// TIA Portal V19 export
VAR_GLOBAL   // PLC tag table "D19"
   D19_Lp_EntryReq_LB321 AT %Q250.2 : Bool;   // 261SH1
   D19_Lp_SafetyReset_LB321 AT %Q250.3 : Bool;   // 261SH2
   D19_Pb_EntryReq_LB321 AT %I250.5 : Bool;   // 261SH1
   D19_Pb_SafetyReset_LB321 AT %I250.6 : Bool;   // 261SH2
   D19_Comando_Elettroserratura AT %Q250.0 : Bool;   // 26102
   D19_Funzione_AUX_Elettroserratura AT %Q250.1 : Bool;   // 26105
   D19_Cancello_Chiuso AT %I250.3 : Bool;   // 26101
   D19_Cancello_Bloccato AT %I250.4 : Bool;   // 26103
   D19_Ls_Os1 AT %I1300.1 : Bool;   // 250DI1 - 261A1
   D19_Ls_Os2 AT %I1300.5 : Bool;   // 250DI5 - 261A1
END_VAR
